INTERFACE I_Motor EXTENDS  __System.IQueryInterface

METHOD Start : BOOL
VAR_INPUT
	
END_VAR
END_METHOD

METHOD Stop : BOOL
VAR_INPUT
	
END_VAR
END_METHOD

END_INTERFACE

(* stored: Version 1.1.0.1, ProductVersion 3.1.4024.16
   Itf I_Motor: Id {9bb9b095-fad3-46a6-a9e2-b966936afb4f}
   Method Start: Id {0ca28784-1984-47b6-910a-ad2c4af38d27}
   Method Stop: Id {64cf7e4a-8a39-4018-97e1-040a672ec88a} *)
